INTERFACE I_Component EXTENDS Calls.I_Arg

END_INTERFACE

(* stored: Version 1.1.0.1
   Itf I_Component: Id {a5dfd892-699d-492b-8b5f-c91d5ccba624} *)
